PROGRAM POU_SawLengthStop
VAR
	requiredSawingLength : INT;
	sawingStopPos: int;
	posReached : BOOL;	
	movingSpeed: INT := 20; // mm/s
	metalAgainstStop: BOOL;
END_VAR

requiredSawingLength := gvl.requiredSawingLength;

IF gvl.startButtonLengthStop THEN
	IF requiredSawingLength = sawingStopPos THEN
		posReached := TRUE;
	ELSE
		sawingStopPos := pou_moveToPos(actualPos := sawingStopPos, requiredPos := requiredSawingLength, speed := movingSpeed);
	END_IF
END_IF

IF metalAgainstStop THEN
	gvl.metalIsToStop := TRUE;
END_IF

END_PROGRAM

(* stored: Version 1.1.0.1, ProductVersion 3.1.4024.12
   POU POU_SawLengthStop: Id {b0fa660f-49cd-4e94-aea0-da98159bb3ad}, SpecialFunc None *)
